// TIA Portal project "Grupo3" (V19)

(* hardware
DEVICE "S7-1200 station_1"  S7-1200 Station
   slot 0: "Rack_0"  S7-1200 Rack  Rack  V1.0
   slot 1: "PLC_1"  CPU 1215C AC/DC/Rly  6ES7 215-1BG40-0XB0  V4.5
*)

// ===== PLC "PLC_1"  CPU 1215C AC/DC/Rly =====

VAR_GLOBAL   // PLC tag table "Default tag table"
   "START" AT %I0.0 : Bool;
   "STOP" AT %I0.1 : Bool;
   "SENSOR" AT %I0.2 : Bool;
   "SELETOR1" AT %I0.3 : Bool;
   "SELETOR2" AT %I0.4 : Bool;
   "SELETOR3" AT %I0.5 : Bool;
   "EMERGENCIA" AT %I0.6 : Bool;
   "AUTO" AT %I0.7 : Bool;
   "TAPETE" AT %Q0.0 : Bool;
   "FORNO" AT %Q0.1 : Bool;
   "SINAL" AT %Q0.2 : Bool;
   "D0" AT %MB2 : Byte;
   "D1" AT %MB3 : Byte;
   "D2" AT %MB4 : Byte;
   "Timer" AT %MB5 : Byte;
END_VAR

ORGANIZATION_BLOCK "Main"   // OB1, LAD, ProgramCycle
TITLE = "Main Program Sweep (Cycle)"
{ S7_Optimized_Access := 'TRUE' }
VERSION : 0.1
   VAR_INPUT
      Initial_Call : Bool;   // Initial call of this OB
      Remanence : Bool;   // =True, if remanent data are available
   END_VAR
BEGIN
END_ORGANIZATION_BLOCK